// TIA Portal V18 export
ORGANIZATION_BLOCK "Cyclic interrupt_comms_50ms"   // OB30, FBD, CyclicInterrupt
{ S7_Optimized_Access := 'TRUE' }
VERSION : 0.1
// stored: AutoNumber true, IsIECCheckEnabled false, SetENOAutomatically false
   VAR_INPUT
      Initial_Call : Bool;
      Event_Count : Int;
   END_VAR
BEGIN

REGION Network 1
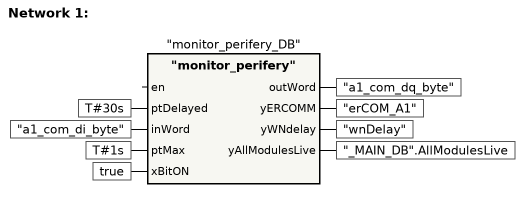
   "monitor_perifery_DB"(ptDelayed := T#30s,   // "monitor_perifery"
                         inWord := "a1_com_di_byte",
                         ptMax := T#1s,
                         xBitON := true,
                         outWord => "a1_com_dq_byte",
                         yERCOMM => "erCOM_A1",
                         yWNdelay => "wnDelay",
                         yAllModulesLive => "_MAIN_DB".AllModulesLive);
END_REGION
END_ORGANIZATION_BLOCK
